(*

## Short summary
This class provides assert statements for ``CNM_AbstractObject.IObjects``  

.. <legal notes>

legal notes
=================
| SPDX-FileCopyrightText: © 2022 ekvip automation GmbH <info@ekvip.de>
| SPDX-License-Identifier: Apache-2.0
| For details check: Apache-2.0_

.. _Apache-2.0: https://www.apache.org/licenses/LICENSE-2.0

.. </legal notes>



*)

{attribute 'reflection'}
FUNCTION_BLOCK INTERNAL ObjectAssertions EXTENDS AbstractAssertion IMPLEMENTS IObjectAssertions
VAR
	(* injected comperator *)
	comperator	: CNM_AbstractObject.IComparator;
END_VAR

(*

## Short summary
This abstract property returns the class name of the concrete object, 
It's for debugging purpose

.. <legal notes>

legal notes
=================
| SPDX-FileCopyrightText: © 2022 ekvip automation GmbH <info@ekvip.de>
| SPDX-License-Identifier: Apache-2.0
| For details check: Apache-2.0_

.. _Apache-2.0: https://www.apache.org/licenses/LICENSE-2.0

.. </legal notes>

*)

PROPERTY className :CNM_AbstractObject.ClassName
GET
className := 'CNM_Assertor.ObjectAssertions';
END_GET
END_PROPERTY

(*

## Short summary
This assertion method checks if ``object`` is after in order to ``objectToCompare``

.. <legal notes>

legal notes
=================
| SPDX-FileCopyrightText: © 2022 ekvip automation GmbH <info@ekvip.de>
| SPDX-License-Identifier: Apache-2.0
| For details check: Apache-2.0_

.. _Apache-2.0: https://www.apache.org/licenses/LICENSE-2.0

.. </legal notes>



*)

METHOD isAfterInOrderTo
VAR_INPUT
	(* object which should be tested *)
	object			:CNM_AbstractObject.IObject;
	(* comparative object *)
	objectToCompare	:CNM_AbstractObject.IObject;
	(* message if the assertion is false *)
	message			:AssertMessage;
END_VAR
IF (THIS^.isObjectNull(THIS^.comperator)) THEN
	IF (THIS^.isObjectValid(object)) THEN
		IF (object.compareTo(objectToCompare) <> CNM_ReturnTypes.ComparationResult.GREATER) THEN
			THIS^.assertionWasWrong(message, THIS^.getDebugInfo('isAfterInOrderTo'));
		END_IF
	ELSIF (THIS^.isObjectValid(objectToCompare)) THEN
		IF (objectToCompare.compareTo(object) >= CNM_ReturnTypes.ComparationResult.EQUAL) THEN
			THIS^.assertionWasWrong(message, THIS^.getDebugInfo('isAfterInOrderTo'));
		END_IF
	ELSE	
		THIS^.assertionWasWrong(message, THIS^.getDebugInfo('isAfterInOrderTo'));
	END_IF
ELSIF (
	THIS^.comperator.compare(object, objectToCompare)
	<> CNM_ReturnTypes.ComparationResult.GREATER
) THEN
	THIS^.assertionWasWrong(message, THIS^.getDebugInfo('isAfterInOrderTo'));
END_IF
END_METHOD

(*

## Short summary
This assertion method checks if ``object``
is at the same position in the sequence as ``objectToCompare``

.. <legal notes>

legal notes
=================
| SPDX-FileCopyrightText: © 2022 ekvip automation GmbH <info@ekvip.de>
| SPDX-License-Identifier: Apache-2.0
| For details check: Apache-2.0_

.. _Apache-2.0: https://www.apache.org/licenses/LICENSE-2.0

.. </legal notes>



*)

METHOD isEqualInOrderTo
VAR_INPUT
	(* object which should be tested *)
	object			:CNM_AbstractObject.IObject;
	(* comparative object *)
	objectToCompare	:CNM_AbstractObject.IObject;
	(* message if the assertion is false *)
	message			:AssertMessage;
END_VAR
IF (THIS^.isObjectNull(THIS^.comperator)) THEN
	IF (THIS^.isObjectValid(object)) THEN
		IF (object.compareTo(objectToCompare) <> CNM_ReturnTypes.ComparationResult.EQUAL) THEN
			THIS^.assertionWasWrong(message, THIS^.getDebugInfo('isEqualInOrderTo'));
		END_IF
	ELSIF (THIS^.isObjectValid(objectToCompare)) THEN
		IF (objectToCompare.compareTo(object) <> CNM_ReturnTypes.ComparationResult.EQUAL) THEN
			THIS^.assertionWasWrong(message, THIS^.getDebugInfo('isEqualInOrderTo'));
		END_IF
	END_IF
ELSIF (
	THIS^.comperator.compare(object, objectToCompare)
	<> CNM_ReturnTypes.ComparationResult.EQUAL
) THEN
	THIS^.assertionWasWrong(message, THIS^.getDebugInfo('isEqualInOrderTo'));
END_IF
END_METHOD

(*

## Short summary
This assertion method checks if ``object`` is ``objectToCompare``

.. <legal notes>

legal notes
=================
| SPDX-FileCopyrightText: © 2022 ekvip automation GmbH <info@ekvip.de>
| SPDX-License-Identifier: Apache-2.0
| For details check: Apache-2.0_

.. _Apache-2.0: https://www.apache.org/licenses/LICENSE-2.0

.. </legal notes>



*)

METHOD isEqualTo
VAR_INPUT
	(* object which should be tested *)
	object			:CNM_AbstractObject.IObject;
	(* comparative object *)
	objectToCompare	:CNM_AbstractObject.IObject;
	(* message if the assertion is false *)
	message			:AssertMessage;
END_VAR
IF (THIS^.isObjectValid(object)) THEN
	IF (NOT object.isEqual(objectToCompare)) THEN
		THIS^.assertionWasWrong(message, THIS^.getDebugInfo('isEqualTo'));
	END_IF
ELSIF (THIS^.isObjectValid(objectToCompare)) THEN
	THIS^.assertionWasWrong(message, THIS^.getDebugInfo('isEqualTo'));
END_IF
END_METHOD

(*

## Short summary
This assertion method checks if ``object`` is not ``objectToCompare``

.. <legal notes>

legal notes
=================
| SPDX-FileCopyrightText: © 2022 ekvip automation GmbH <info@ekvip.de>
| SPDX-License-Identifier: Apache-2.0
| For details check: Apache-2.0_

.. _Apache-2.0: https://www.apache.org/licenses/LICENSE-2.0

.. </legal notes>



*)

METHOD isNotEqualTo
VAR_INPUT
	(* object which should be tested *)
	object			:CNM_AbstractObject.IObject;
	(* comparative object *)
	objectToCompare	:CNM_AbstractObject.IObject;
	(* message if the assertion is false *)
	message			:AssertMessage;
END_VAR
IF (THIS^.isObjectValid(object)) THEN
	IF (object.isEqual(objectToCompare)) THEN
		THIS^.assertionWasWrong(message, THIS^.getDebugInfo('isNotEqualTo'));
	END_IF
ELSIF (THIS^.isObjectNull(objectToCompare)) THEN
	THIS^.assertionWasWrong(message, THIS^.getDebugInfo('isNotEqualTo'));
END_IF
END_METHOD

(*

## Short summary
This assertion method checks if ``object`` is NULL

.. <legal notes>

legal notes
=================
| SPDX-FileCopyrightText: © 2022 ekvip automation GmbH <info@ekvip.de>
| SPDX-License-Identifier: Apache-2.0
| For details check: Apache-2.0_

.. _Apache-2.0: https://www.apache.org/licenses/LICENSE-2.0

.. </legal notes>



*)

METHOD objectIsNull
VAR_INPUT
	(* object which should be tested *)
	object	:CNM_AbstractObject.IObject;
	(* message if the assertion is false *)
	message	:AssertMessage;
END_VAR
IF (THIS^.isObjectValid(object)) THEN
	THIS^.assertionWasWrong(message, THIS^.getDebugInfo('objectIsNull'));
END_IF
END_METHOD

(*

## Short summary
This assertion method checks if ``object`` is not NULL

.. <legal notes>

legal notes
=================
| SPDX-FileCopyrightText: © 2022 ekvip automation GmbH <info@ekvip.de>
| SPDX-License-Identifier: Apache-2.0
| For details check: Apache-2.0_

.. _Apache-2.0: https://www.apache.org/licenses/LICENSE-2.0

.. </legal notes>



*)

METHOD objectIsValid
VAR_INPUT
	(* object which should be tested *)
	object	:CNM_AbstractObject.IObject;
	(* message if the assertion is false *)
	message	:AssertMessage;
END_VAR
IF (NOT THIS^.isObjectValid(object)) THEN
	THIS^.assertionWasWrong(message, THIS^.getDebugInfo('objectIsValid'));
END_IF
END_METHOD

(*

## Short summary
This assertion method checks if ``object``
precedes in sequence to ``objectToCompare``

.. <legal notes>

legal notes
=================
| SPDX-FileCopyrightText: © 2022 ekvip automation GmbH <info@ekvip.de>
| SPDX-License-Identifier: Apache-2.0
| For details check: Apache-2.0_

.. _Apache-2.0: https://www.apache.org/licenses/LICENSE-2.0

.. </legal notes>



*)

METHOD precedesInOrderTo
VAR_INPUT
	(* object which should be tested *)
	object			:CNM_AbstractObject.IObject;
	(* comparative object *)
	objectToCompare	:CNM_AbstractObject.IObject;
	(* message if the assertion is false *)
	message			:AssertMessage;
END_VAR
IF (THIS^.isObjectNull(THIS^.comperator)) THEN
	IF (THIS^.isObjectValid(object)) THEN
		IF (object.compareTo(objectToCompare) <> CNM_ReturnTypes.ComparationResult.SMALLER) THEN
			THIS^.assertionWasWrong(message, THIS^.getDebugInfo('precedesInOrderTo'));
		END_IF
	ELSIF (THIS^.isObjectValid(objectToCompare)) THEN
		IF (objectToCompare.compareTo(object) <= CNM_ReturnTypes.ComparationResult.EQUAL) THEN
			THIS^.assertionWasWrong(message, THIS^.getDebugInfo('precedesInOrderTo'));
		END_IF
	ELSE	
		THIS^.assertionWasWrong(message, THIS^.getDebugInfo('precedesInOrderTo'));
	END_IF
ELSIF (
	THIS^.comperator.compare(object, objectToCompare)
	<> CNM_ReturnTypes.ComparationResult.SMALLER
) THEN
	THIS^.assertionWasWrong(message, THIS^.getDebugInfo('precedesInOrderTo'));
END_IF
END_METHOD

(*

## Short summary
This allows you to set your own comperator for the methods
`IObjectAssertions.precedesInOrderTo`  
`IObjectAssertions.isEqualInOrderTo`  
`IObjectAssertions.isAfterInOrderTo`
to clear the comperator again, just call it with 0: ``foo.setComperator(comperator := 0);``

.. <legal notes>

legal notes
=================
| SPDX-FileCopyrightText: © 2022 ekvip automation GmbH <info@ekvip.de>
| SPDX-License-Identifier: Apache-2.0
| For details check: Apache-2.0_

.. _Apache-2.0: https://www.apache.org/licenses/LICENSE-2.0

.. </legal notes>



*)

METHOD setComperator
VAR_INPUT
	(* comperator to inject *)
	comperator	:CNM_AbstractObject.IComparator := 0;
END_VAR
THIS^.comperator := comperator;
END_METHOD

END_FUNCTION_BLOCK

(* stored: Version 1.1.0.1, ProductVersion 3.1.4026.11
   POU ObjectAssertions: Id {6b0104dc-0fa5-4796-b05c-cc0271c4c02e}, SpecialFunc None
   Property className: Id {76a4cba8-ada8-4bf0-b8ac-6f3bcb8eeac1}
   Get Get: Id {01f12f0f-96cc-4167-bb44-c74436b4326a}
   Method isAfterInOrderTo: Id {b7a0129b-14a0-464a-8c6e-3e425c5c2dc8}
   Method isEqualInOrderTo: Id {11d54115-1f87-4097-98bc-7287b9134de6}
   Method isEqualTo: Id {0684d09c-0456-4ad1-9e66-4e9998502043}
   Method isNotEqualTo: Id {db7266fe-1971-4010-8539-fb86bedb9744}
   Method objectIsNull: Id {f4944f04-968a-4e94-8665-33487c8a9b2b}
   Method objectIsValid: Id {48a1a2d3-5740-4e3e-9864-08b0175b7f37}
   Method precedesInOrderTo: Id {ee776579-a813-496b-9c62-857e1ce9e857}
   Method setComperator: Id {63bdbad0-6e7b-42cd-b3d0-55596e213964} *)
